FUNCTION_BLOCK CappingStationCtrl (* Template for an empty basic function block *)
  (* Standard: 61499-2 *)
  (* Version 1.0, 2018-09-15, az *)
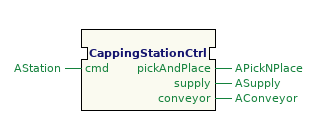
  SOCKETS
    cmd : AStation;
  END_SOCKETS
  PLUGS
    pickAndPlace : APickNPlace;
    supply : ASupply;
    conveyor : AConveyor;
  END_PLUGS
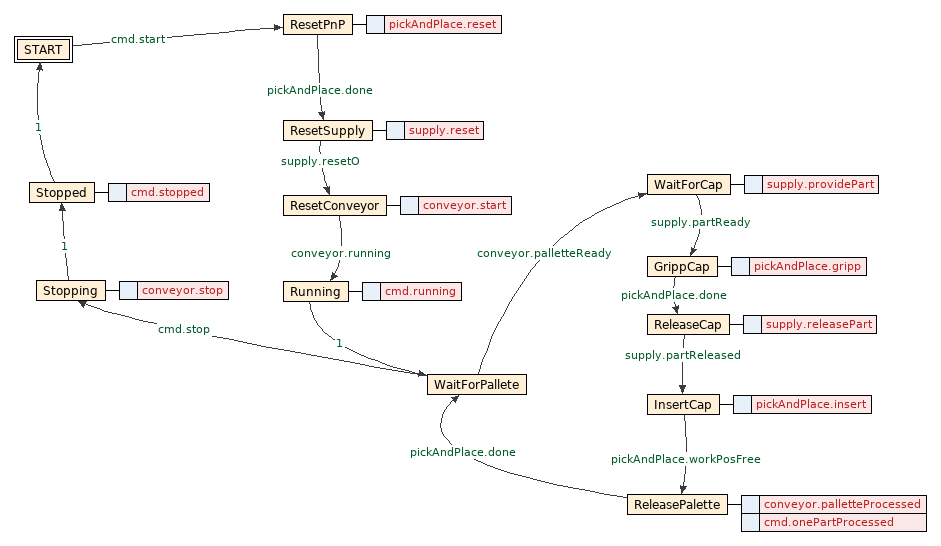
  EC_STATES
    START; (* Initial State *)
    ResetPnP : -> pickAndPlace.reset;
    ResetSupply : -> supply.reset;
    ResetConveyor : -> conveyor.start;
    Running : -> cmd.running;
    Stopping : -> conveyor.stop;
    Stopped : -> cmd.stopped;
    WaitForPallete;
    WaitForCap : -> supply.providePart;
    GrippCap : -> pickAndPlace.gripp;
    ReleaseCap : -> supply.releasePart;
    InsertCap : -> pickAndPlace.insert;
    ReleasePalette : -> conveyor.palletteProcessed, -> cmd.onePartProcessed;
  END_STATES
  EC_TRANSITIONS
    START TO ResetPnP := cmd.start;
    ResetPnP TO ResetSupply := pickAndPlace.done;
    ResetSupply TO ResetConveyor := supply.resetO;
    ResetConveyor TO Running := conveyor.running;
    Stopped TO START := 1;
    Stopping TO Stopped := 1;
    WaitForPallete TO Stopping := cmd.stop;
    Running TO WaitForPallete := 1;
    WaitForPallete TO WaitForCap := conveyor.palletteReady;
    WaitForCap TO GrippCap := supply.partReady;
    GrippCap TO ReleaseCap := pickAndPlace.done;
    InsertCap TO ReleasePalette := pickAndPlace.workPosFree;
    ReleaseCap TO InsertCap := supply.partReleased;
    ReleasePalette TO WaitForPallete := pickAndPlace.done;
  END_TRANSITIONS
END_FUNCTION_BLOCK
